TYPE ST_InputTable_MitsubishiWithWheelHouse EXTENDS ST_InputTable_Mitsubishi :
STRUCT
	arWheelhouseInput : ARRAY[1..400] OF BOOL;
END_STRUCT
END_TYPE

(* stored: Version 1.1.0.1, ProductVersion 3.1.4024.13
   DUT ST_InputTable_MitsubishiWithWheelHouse: Id {344c3661-a21b-4ecd-a97c-8ac93ba790e8} *)
